// TwinCAT 3 PLC project PLC
// ProgramVersion: 3.1.4024.0
// libraries:
//   Tc2_MC2, * (Beckhoff Automation GmbH)
//   Tc2_Standard, * (Beckhoff Automation GmbH)
//   Tc2_System, * (Beckhoff Automation GmbH)
//   Tc3_Module, * (Beckhoff Automation GmbH)
//   VisuDialogs, * (System)
//   VisuSymbols,3.5.10.0,System
// project tree:
//   / Gestore di visualizzazione.TcVMO (not stored), GlobalTextList.TcGTLO, PlcTask.TcTTO (not stored)
//   GVLs/ GVL.TcGVL
//   POUs/ MAIN.TcPOU
//   VISUs/ Visualization.TcVIS
// real-time tasks:
//   TASK PlcTask: cycle T#10ms, priority 20, ADS port 350
// motion (NC):
//   TASK NC-Task 1 SAF: cycle T#2ms, priority 4, ADS port 501
//   TASK NC-Task 1 SVB: cycle T#10ms, priority 8, ADS port 511
//   AXIS Asse 1 (id 1)
//     OtherSettings: AllowMotionCmdToSlave=true
//     encoder EncType=1
//       Inc: RefSoftSyncMask=#x0000ffff
//     drive DrvType=24
//       Analog: TorqueSetpointScale=10, ScaleFactorActTorque=0.1
//       TimeComp: TaskDelayCycles=1
//     controller CtrType=1
//       CtrPara: PriorControlFactor=1
//         Observer: BandWidth=20
// I/O:
//   DEVICE Dispositivo 1 (EtherCAT), AmsNetId 192.168.10.25.2.1
//     Terminale 1 (EK1200) [EK1200-5000 EtherCAT Power supply (2A E-Bus)]
//       Terminale 2 (EL1008) [EL1008 8Ch. Dig. Input 24V, 3ms]
//       Terminale 3 (EL2008) [EL2008 8Ch. Dig. Output 24V, 0.5A]
//       Terminale 4 (EL3064) [EL3064 4Ch. Ana. Input 0-10V]
//       Terminale 5 (EL4002) [EL4002 2Ch. Ana. Output 0-10V, 12bit]
//       Terminale 6 (EL3202) [EL3202 2Ch. Ana. Input PT100 (RTD)]
//       Terminale 7 (EL4022) [EL4022 2Ch. Ana. Output 4-20mA, 12bit]
//       Terminale 8 (EL7047) [EL7047 1Ch. Stepper motor output stage (50V, 5A)]
//       Terminale 9 (EL9011) [EL9011 End Terminal]
// variable links:
//   NC-Task 1 SAF/Axes/Asse 1 <-> Device 1 (EtherCAT)/Term 1 (EK1200)/Term 8 (EL7047)
//     Drive/Inputs/In/nState1 @bit 3 <-> STM Status/Status/Error
//     Drive/Inputs/In/nState1 @bit 7 <-> STM Status/Status/Motor stall
//     Drive/Inputs/In/nState1 @bit 5 <-> STM Status/Status/Moving negative
//     Drive/Inputs/In/nState1 @bit 4 <-> STM Status/Status/Moving positive
//     Drive/Inputs/In/nState1 @bit 1 <-> STM Status/Status/Ready
//     Drive/Inputs/In/nState1 <-> STM Status/Status/Ready to enable
//     Drive/Inputs/In/nState1 @bit 6 <-> STM Status/Status/Torque reduced
//     Drive/Inputs/In/nState1 @bit 2 <-> STM Status/Status/Warning
//     Drive/Inputs/In/nState2 @bit 3 <-> STM Status/Status/Digital input 1
//     Drive/Inputs/In/nState2 @bit 4 <-> STM Status/Status/Digital input 2
//     Drive/Inputs/In/nState2 @bit 5 <-> STM Status/Status/Sync error
//     Drive/Inputs/In/nState2 @bit 7 <-> STM Status/Status/TxPDO Toggle
//     Drive/Inputs/In/nState4 @bit 1 <-> WcState/InputToggle
//     Drive/Inputs/In/nState4 <-> WcState/WcState
//     Drive/Outputs/Out/nCtrl1 <-> STM Control/Control/Enable
//     Drive/Outputs/Out/nCtrl1 @bit 2 <-> STM Control/Control/Reduce torque
//     Drive/Outputs/Out/nCtrl1 @bit 1 <-> STM Control/Control/Reset
//     Drive/Outputs/Out/nCtrl2 @bit 3 <-> STM Control/Control/Digital output 1
//     Drive/Outputs/Out/nDataOut2[0] <-> STM Velocity/Velocity
//     Enc/Inputs/In/nDataIn1[0] <-> ENC Status compact/Counter value
//     Enc/Inputs/In/nDataIn2[0] <-> ENC Status compact/Latch value
//     Enc/Inputs/In/nState1 @bit 4 <-> ENC Status compact/Status/Counter overflow
//     Enc/Inputs/In/nState1 @bit 3 <-> ENC Status compact/Status/Counter underflow
//     Enc/Inputs/In/nState1 @bit 7 <-> ENC Status compact/Status/Extrapolation stall
//     Enc/Inputs/In/nState1 <-> ENC Status compact/Status/Latch C valid
//     Enc/Inputs/In/nState1 @bit 1 <-> ENC Status compact/Status/Latch extern valid
//     Enc/Inputs/In/nState1 @bit 2 <-> ENC Status compact/Status/Set counter done
//     Enc/Inputs/In/nState2 @bit 4 <-> ENC Status compact/Status/Status of extern latch
//     Enc/Inputs/In/nState2 <-> ENC Status compact/Status/Status of input A
//     Enc/Inputs/In/nState2 @bit 1 <-> ENC Status compact/Status/Status of input B
//     Enc/Inputs/In/nState2 @bit 2 <-> ENC Status compact/Status/Status of input C
//     Enc/Inputs/In/nState2 @bit 5 <-> ENC Status compact/Status/Sync error
//     Enc/Inputs/In/nState2 @bit 7 <-> ENC Status compact/Status/TxPDO Toggle
//     Enc/Inputs/In/nState4 @bit 1 <-> WcState/InputToggle
//     Enc/Inputs/In/nState4 <-> WcState/WcState
//     Enc/Outputs/Out/nCtrl1 <-> ENC Control compact/Control/Enable latch C
//     Enc/Outputs/Out/nCtrl1 @bit 3 <-> ENC Control compact/Control/Enable latch extern on negative edge
//     Enc/Outputs/Out/nCtrl1 @bit 1 <-> ENC Control compact/Control/Enable latch extern on positive edge
//     Enc/Outputs/Out/nCtrl1 @bit 2 <-> ENC Control compact/Control/Set counter
//     Enc/Outputs/Out/nDataOut1[0] <-> ENC Control compact/Set counter value
//   PLC/PLC Instance <-> NC-Task 1 SAF/Axes/Asse 1
//     PlcTask Inputs/GVL.axis.NcToPlc <-> Outputs/ToPlc
//     PlcTask Outputs/GVL.axis.PlcToNc <-> Inputs/FromPlc

// ---- GVLs/GVL.TcGVL
{attribute 'qualified_only'}
VAR_GLOBAL
	bStartButton: BOOL;
	bStopButton: BOOL;
	fVelocity: REAL;
	fAccelleration: REAL;
	
	//Output
	nMotorPosition: LREAL;
	bMotorEnabled: BOOL;
	bMotorForward: BOOL;
	bMotorBackwards: BOOL;
	
	//Internal
	axis: AXIS_REF;
	fBJog: MC_Jog;
	fBPower: MC_Power;
END_VAR

// ---- POUs/MAIN.TcPOU
PROGRAM MAIN
VAR
END_VAR

Comandi();
Motore();

ACTION Comandi:
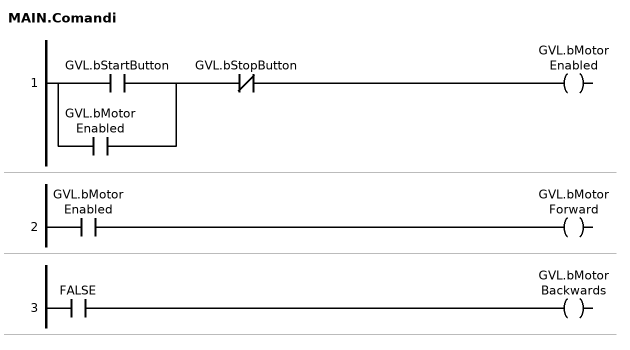
// NETWORK 1
GVL.bMotorEnabled := (GVL.bStartButton OR GVL.bMotorEnabled) AND NOT GVL.bStopButton;

// NETWORK 2
GVL.bMotorForward := GVL.bMotorEnabled;

// NETWORK 3
GVL.bMotorBackwards := FALSE;
END_ACTION

ACTION Motore:
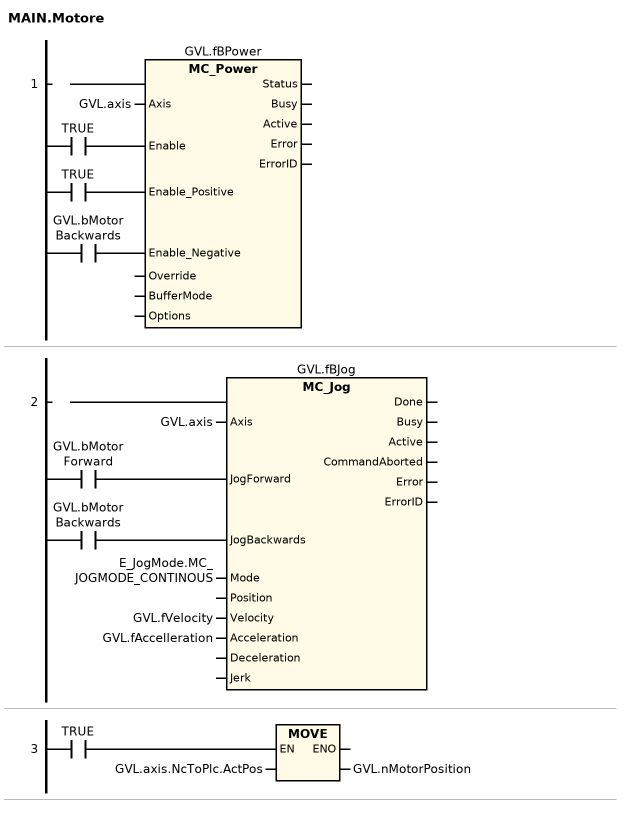
// NETWORK 1
GVL.fBPower(
    Axis := GVL.axis,
    Enable := TRUE,
    Enable_Positive := TRUE,
    Enable_Negative := GVL.bMotorBackwards); // MC_Power

// NETWORK 2
GVL.fBJog(
    Axis := GVL.axis,
    JogForward := GVL.bMotorForward,
    JogBackwards := GVL.bMotorBackwards,
    Mode := E_JogMode.MC_JOGMODE_CONTINOUS,
    Velocity := GVL.fVelocity,
    Acceleration := GVL.fAccelleration); // MC_Jog

// NETWORK 3
GVL.nMotorPosition := GVL.axis.NcToPlc.ActPos;
END_ACTION

END_PROGRAM

// ---- GlobalTextList.TcGTLO
TEXTLIST GlobalTextList
  941 = '%d'
  392 = '%f'
  426 = 'Accelerazione attuale [mm/s]'
  676 = 'Accelerazione attuale [mm/s^2]'
  581 = 'Accelerazione [mm/s^2]'
  945 = 'Posizione [mm]'
  294 = 'START'
  404 = 'STOP'
  834 = 'Velocità'
  781 = 'Velocità attuale [mm/s]'
  370 = 'Velocità [mm/s]'
END_TEXTLIST

// ---- VISUs/Visualization.TcVIS
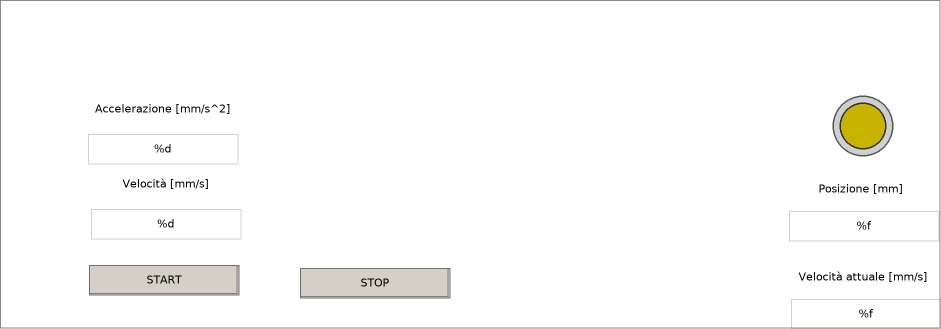
VISUALIZATION Visualization  // 941x329
    Lamp1 (828,91 70x70), variable: GVL.bMotorForward, style: Lamp-Lamp1-Yellow
    Button (89,265 150x30), "START"
        tap GVL.bStartButton
    Button (300,268 150x30), "STOP"
        tap GVL.bStopButton
    Textfield (789,211 150x30), "%f", text variable: GVL.nMotorPosition
    Textfield (91,209 150x30), "%d", text variable: GVL.fVelocity
        OnMouseClick: write the text variable via Default, min 0, max 7000, title "Velocità"
    Label (91,169 150x30), "Velocità [mm/s]"
    Label (786,174 150x30), "Posizione [mm]"
    Textfield (791,299 150x30), "%f", text variable: GVL.axis.NcToPlc.ActVelo
    Label (788,262 150x30), "Velocità attuale [mm/s]"
    Textfield (88,134 150x30), "%d", text variable: GVL.fAccelleration
        OnMouseClick: write the text variable via Default, min 0, max 500, title "Velocità"
    Label (88,94 150x30), "Accelerazione [mm/s^2]"
END_VISUALIZATION
